FUNCTION TryConvert_LWORD_TO_INT : BOOL
VAR_INPUT
	in : LWORD;
	out : REFERENCE TO INT;
END_VAR

IF in > DatatypeLimits.MAX_VALUE_OF_LWORD_WHICH_CAN_BE_HELD_IN_A_INT THEN
	RETURN;
END_IF

out := LWORD_TO_INT(in);
TryConvert_LWORD_TO_INT := TRUE;

END_FUNCTION

(* stored: Version 1.1.0.1, ProductVersion 3.1.4024.12
   POU TryConvert_LWORD_TO_INT: Id {779aeea0-1217-4daf-b335-16bb3a6bc011}, SpecialFunc None *)
